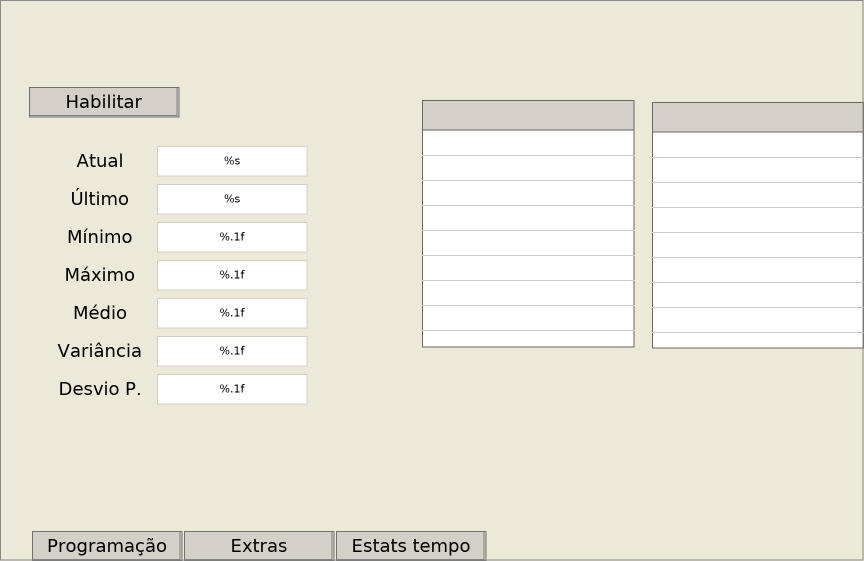
VISUALIZATION EstatisticaTempo  // 864x561
    Button (32,531 150x30), "Programação"
        OnMouseClick: change screen: Visualization
    Button (184,531 150x30), "Extras"
        OnMouseClick: change screen: FuncoesExtras
    Button (336,531 150x30), "Estats tempo"
        OnMouseClick: change screen: EstatisticaTempo
    Table (422,100 212x247), data array: prgTimeStatistics.lastTimes
        p3854506369: prgTimeStatistics.lastTimes[INDEX]
        p2232123230: Últimos tempos (T)
    Table (652,102 212x246), data array: prgTimeStatistics.arLastTimes
        p3854506369: prgTimeStatistics.arLastTimes[INDEX]
        p2232123230: Últimos tempos (s)
    Button (29,87 150x30), "Habilitar"
        toggle prgTimeStatistics.enableTimeCount
    Label (40,146 120x30), "Atual"
    Label (40,184 120x30), "Último"
    Label (40,222 120x30), "Mínimo"
    Label (40,260 120x30), "Máximo"
    Label (40,298 120x30), "Médio"
    Label (40,336 120x30), "Variância"
    Label (40,374 120x30), "Desvio P."
    Textfield (157,146 150x30), "%s", text variable: prgTimeStatistics.lastTimeStats.currTime
    Textfield (157,184 150x30), "%s", text variable: prgTimeStatistics.lastTimeStats.lastTime
    Textfield (157,222 150x30), "%.1f", text variable: prgTimeStatistics.stats.minimum
    Textfield (157,260 150x30), "%.1f", text variable: prgTimeStatistics.stats.maximum
    Textfield (157,298 150x30), "%.1f", text variable: prgTimeStatistics.stats.avg
    Textfield (157,336 150x30), "%.1f", text variable: prgTimeStatistics.stats.variance
    Textfield (157,374 150x30), "%.1f", text variable: prgTimeStatistics.stats.standardDeviation
END_VISUALIZATION

(* stored: Version 1.1.0.1, ProductVersion 3.1.4024.11
   Visu EstatisticaTempo: Id {139b8c2c-dc94-44c5-8aec-aa2878dd0bed} *)
